(* IEC 61131-3 sources: plc-home-automation/home_automation/lighting_heating_updated/src/alarm, 4 files *)

(* ---- AlarmGlobals.st ---- *)
VAR_GLOBAL CONSTANT

   C_FRONT_DOOR_OPENING : INT     := 1;
   C_GARAGE_DOOR_OPENING : UINT   := 2;
   C_HALL_ZONE : UINT             := 4;
   C_GARAGE_ZONE : UINT           := 5;
   C_KITCHEN_ZONE : UINT          := 6;
   C_LIVING_ROOM_ZONE : UINT      := 7;
   C_BEDROOM_ZONE : UINT          := 8;
   C_DOWNSTAIRS_BATH_ZONE : UINT  := 9;
   C_HALLWAY_ZONE : UINT          := 10;
   C_CHILDRENS_ROOM_3_ZONE : UINT := 11;
   C_CHILDRENS_ROOM_1_ZONE : UINT := 12;
   C_CHILDRENS_ROOM_2_ZONE : UINT := 13;
   C_UPSTAIRS_BATH_ZONE : UINT    := 14;
   C_WC_ZONE : UINT               := 15;
   C_BOILER_ZONE : UINT           := 16;

   C_UNCONNECTED_NO_OP : UINT     := 3;

   C_ALARM_ZONES : UINT           := 16;
END_VAR

VAR_GLOBAL
    PARADOX_COM : fbPAR_DIG_EVOsystem;
    PARADOX_DATA : T_PAR_DIG_EVO_SYSTEM_DATA;
    ALARM_ZONES_INACTIVITY : ARRAY [1 .. C_ALARM_ZONES] OF BOOL;
    ALARM_ZONES_SABOTAGE : ARRAY [1 .. C_ALARM_ZONES] OF BOOL;
    ALARM_ZONES_ERROR : ARRAY [1 .. C_ALARM_ZONES] OF BOOL;
    ALARM_ACTIVE : BOOL;

    PRESENCE_BASED_HEATING_CONTROL : BOOL   := true;
    PRESENCE_BASED_HOT_WATER_CONTROL : BOOL := true;
    PRESENCE_BASED_HEATING_ENABLE : BOOL    := false;
    PRESENCE_BASED_HOT_WATER_ENABLE : BOOL  := false;

    AWAY_TIMER: TON;

    TIME_AWAY_SHORT : TIME     := T#20m;
    TIME_AWAY_LONG : TIME      := T#60m;
    GONE_FOR_5_SECONDS : BOOL  := FALSE; // for debugging purposes
    GONE_FOR_5_MINUTES : BOOL  := FALSE;
    GONE_FOR_5_HOURS : BOOL    := FALSE;
    GONE_FOR_SHORT_TIME : BOOL := FALSE;
    GONE_FOR_LONG_TIME : BOOL  := FALSE;
END_VAR

FUNCTION awayFromHomeFor : bool
  VAR_INPUT
    awayFor : TIME;  (*Tell me if motion sensors are inactive for that time. Max is 20 days.*)
  END_VAR

  IF(AWAY_TIMER.ET < awayFor) THEN
    awayFromHomeFor := false;
  ELSE
    awayFromHomeFor := true;
  END_IF;

END_FUNCTION

(* ---- AlarmRead.st ---- *)
FUNCTION alarmRead : BOOL

VAR_INPUT
END_VAR

VAR
  inactive_no_operation : BOOL := TRUE;
END_VAR

  PARADOX_COM(chan_code := CH1_uni, max_zone_count := C_ALARM_ZONES, par_system_data := PARADOX_DATA);
  alarmRead := PARADOX_COM.com_ok;

  ALARM_ZONES_INACTIVITY[C_FRONT_DOOR_OPENING] := PARADOX_DATA.zone[C_FRONT_DOOR_OPENING].state;
  ALARM_ZONES_INACTIVITY[C_GARAGE_DOOR_OPENING] := PARADOX_DATA.zone[C_GARAGE_DOOR_OPENING].state;
  ALARM_ZONES_INACTIVITY[C_HALL_ZONE] := PARADOX_DATA.zone[C_HALL_ZONE].state;
  ALARM_ZONES_INACTIVITY[C_GARAGE_ZONE] := PARADOX_DATA.zone[C_GARAGE_ZONE].state;
  ALARM_ZONES_INACTIVITY[C_KITCHEN_ZONE] := PARADOX_DATA.zone[C_KITCHEN_ZONE].state;
  ALARM_ZONES_INACTIVITY[C_LIVING_ROOM_ZONE] := PARADOX_DATA.zone[C_LIVING_ROOM_ZONE].state;
  ALARM_ZONES_INACTIVITY[C_BEDROOM_ZONE] := PARADOX_DATA.zone[C_BEDROOM_ZONE].state;
  ALARM_ZONES_INACTIVITY[C_DOWNSTAIRS_BATH_ZONE] := PARADOX_DATA.zone[C_DOWNSTAIRS_BATH_ZONE].state;
  ALARM_ZONES_INACTIVITY[C_HALLWAY_ZONE] := PARADOX_DATA.zone[C_HALLWAY_ZONE].state;
  ALARM_ZONES_INACTIVITY[C_CHILDRENS_ROOM_3_ZONE] := PARADOX_DATA.zone[C_CHILDRENS_ROOM_3_ZONE].state;
  ALARM_ZONES_INACTIVITY[C_CHILDRENS_ROOM_1_ZONE] := PARADOX_DATA.zone[C_CHILDRENS_ROOM_1_ZONE].state;
  ALARM_ZONES_INACTIVITY[C_CHILDRENS_ROOM_2_ZONE] := PARADOX_DATA.zone[C_CHILDRENS_ROOM_2_ZONE].state;
  ALARM_ZONES_INACTIVITY[C_UPSTAIRS_BATH_ZONE] := PARADOX_DATA.zone[C_UPSTAIRS_BATH_ZONE].state;
  ALARM_ZONES_INACTIVITY[C_WC_ZONE] := PARADOX_DATA.zone[C_WC_ZONE].state;
  ALARM_ZONES_INACTIVITY[C_BOILER_ZONE] := PARADOX_DATA.zone[C_BOILER_ZONE].state;

  ALARM_ZONES_SABOTAGE[C_FRONT_DOOR_OPENING] := PARADOX_DATA.zone[C_FRONT_DOOR_OPENING].tamper;
  ALARM_ZONES_SABOTAGE[C_GARAGE_DOOR_OPENING] := PARADOX_DATA.zone[C_GARAGE_DOOR_OPENING].tamper;
  ALARM_ZONES_SABOTAGE[C_HALL_ZONE] := PARADOX_DATA.zone[C_HALL_ZONE].tamper;
  ALARM_ZONES_SABOTAGE[C_GARAGE_ZONE] := PARADOX_DATA.zone[C_GARAGE_ZONE].tamper;
  ALARM_ZONES_SABOTAGE[C_KITCHEN_ZONE] := PARADOX_DATA.zone[C_KITCHEN_ZONE].tamper;
  ALARM_ZONES_SABOTAGE[C_LIVING_ROOM_ZONE] := PARADOX_DATA.zone[C_LIVING_ROOM_ZONE].tamper;
  ALARM_ZONES_SABOTAGE[C_BEDROOM_ZONE] := PARADOX_DATA.zone[C_BEDROOM_ZONE].tamper;
  ALARM_ZONES_SABOTAGE[C_DOWNSTAIRS_BATH_ZONE] := PARADOX_DATA.zone[C_DOWNSTAIRS_BATH_ZONE].tamper;
  ALARM_ZONES_SABOTAGE[C_HALLWAY_ZONE] := PARADOX_DATA.zone[C_HALLWAY_ZONE].tamper;
  ALARM_ZONES_SABOTAGE[C_CHILDRENS_ROOM_3_ZONE] := PARADOX_DATA.zone[C_CHILDRENS_ROOM_3_ZONE].tamper;
  ALARM_ZONES_SABOTAGE[C_CHILDRENS_ROOM_1_ZONE] := PARADOX_DATA.zone[C_CHILDRENS_ROOM_1_ZONE].tamper;
  ALARM_ZONES_SABOTAGE[C_CHILDRENS_ROOM_2_ZONE] := PARADOX_DATA.zone[C_CHILDRENS_ROOM_2_ZONE].tamper;
  ALARM_ZONES_SABOTAGE[C_UPSTAIRS_BATH_ZONE] := PARADOX_DATA.zone[C_UPSTAIRS_BATH_ZONE].tamper;
  ALARM_ZONES_SABOTAGE[C_WC_ZONE] := PARADOX_DATA.zone[C_WC_ZONE].tamper;
  ALARM_ZONES_SABOTAGE[C_BOILER_ZONE] := PARADOX_DATA.zone[C_BOILER_ZONE].tamper;

  ALARM_ZONES_ERROR[C_FRONT_DOOR_OPENING] := PARADOX_DATA.zone[C_FRONT_DOOR_OPENING].fault;
  ALARM_ZONES_ERROR[C_GARAGE_DOOR_OPENING] := PARADOX_DATA.zone[C_GARAGE_DOOR_OPENING].fault;
  ALARM_ZONES_ERROR[C_HALL_ZONE] := PARADOX_DATA.zone[C_HALL_ZONE].fault;
  ALARM_ZONES_ERROR[C_GARAGE_ZONE] := PARADOX_DATA.zone[C_GARAGE_ZONE].fault;
  ALARM_ZONES_ERROR[C_KITCHEN_ZONE] := PARADOX_DATA.zone[C_KITCHEN_ZONE].fault;
  ALARM_ZONES_ERROR[C_LIVING_ROOM_ZONE] := PARADOX_DATA.zone[C_LIVING_ROOM_ZONE].fault;
  ALARM_ZONES_ERROR[C_BEDROOM_ZONE] := PARADOX_DATA.zone[C_BEDROOM_ZONE].fault;
  ALARM_ZONES_ERROR[C_DOWNSTAIRS_BATH_ZONE] := PARADOX_DATA.zone[C_DOWNSTAIRS_BATH_ZONE].fault;
  ALARM_ZONES_ERROR[C_HALLWAY_ZONE] := PARADOX_DATA.zone[C_HALLWAY_ZONE].fault;
  ALARM_ZONES_ERROR[C_CHILDRENS_ROOM_3_ZONE] := PARADOX_DATA.zone[C_CHILDRENS_ROOM_3_ZONE].fault;
  ALARM_ZONES_ERROR[C_CHILDRENS_ROOM_1_ZONE] := PARADOX_DATA.zone[C_CHILDRENS_ROOM_1_ZONE].fault;
  ALARM_ZONES_ERROR[C_CHILDRENS_ROOM_2_ZONE] := PARADOX_DATA.zone[C_CHILDRENS_ROOM_2_ZONE].fault;
  ALARM_ZONES_ERROR[C_UPSTAIRS_BATH_ZONE] := PARADOX_DATA.zone[C_UPSTAIRS_BATH_ZONE].fault;
  ALARM_ZONES_ERROR[C_WC_ZONE] := PARADOX_DATA.zone[C_WC_ZONE].fault;
  ALARM_ZONES_ERROR[C_BOILER_ZONE] := PARADOX_DATA.zone[C_BOILER_ZONE].fault;

  ALARM_ZONES_INACTIVITY[C_UNCONNECTED_NO_OP] := inactive_no_operation;
  ALARM_ZONES_SABOTAGE[C_UNCONNECTED_NO_OP] := inactive_no_operation;
  ALARM_ZONES_ERROR[C_UNCONNECTED_NO_OP] := inactive_no_operation;

  ALARM_ACTIVE := PARADOX_DATA.part[1].state.armed;

  return;

END_FUNCTION

(* ---- Alarm.st ---- *)
PROGRAM AlarmControl
  VAR_INPUT
  END_VAR
  VAR_OUTPUT
  END_VAR
  VAR
     i: UINT;
     sumActivity : BOOL := FALSE;

     requestOffHeating : BOOL;
     requestOffHotWater : BOOL;

     heatingControl : ChangeOnOff;
     hotWaterControl : ChangeOnOff;

     heatingControllerName : STRING := 'Alarm heating control';
     hotWaterControllerName : STRING := 'Alarm hot water control';
  END_VAR

  alarmRead();

  // Turn on warm water circulation when someone enters through the entrance doors after the alarm cooldown time.
  VIRTUAL_CIRCULATION_SWITCH_IN := GONE_FOR_SHORT_TIME AND
      (NOT ALARM_ZONES_INACTIVITY[C_GARAGE_DOOR_OPENING] OR NOT ALARM_ZONES_INACTIVITY[C_FRONT_DOOR_OPENING]);

  // Detecting if house is no longer occupied or everyone is sleeping
  sumActivity := FALSE;
  FOR i := 1 TO C_ALARM_ZONES DO
     sumActivity := sumActivity OR (NOT ALARM_ZONES_INACTIVITY[i]);
  END_FOR;
  AWAY_TIMER(IN := NOT sumActivity, PT := T#20d);
  GONE_FOR_5_SECONDS  := awayFromHomeFor(awayFor := T#5s);
  GONE_FOR_5_MINUTES  := awayFromHomeFor(awayFor := T#5m);
  GONE_FOR_5_HOURS    := awayFromHomeFor(awayFor := T#5h);
  GONE_FOR_SHORT_TIME := awayFromHomeFor(TIME_AWAY_SHORT);
  GONE_FOR_LONG_TIME  := awayFromHomeFor(TIME_AWAY_LONG);

  requestOffHeating := ((ALARM_ACTIVE AND GONE_FOR_5_MINUTES) OR GONE_FOR_5_HOURS);
  requestOffHotWater:= ((ALARM_ACTIVE AND GONE_FOR_5_MINUTES) OR GONE_FOR_SHORT_TIME);

  IF PRESENCE_BASED_HEATING_CONTROL THEN
     heatingControl(requestOn := NOT requestOffHeating,
         requestOff := requestOffHeating,
         name := heatingControllerName);
     PRESENCE_BASED_HEATING_ENABLE := heatingControl.output;
  END_IF;

  IF PRESENCE_BASED_HOT_WATER_CONTROL THEN
     hotWaterControl(requestOn := NOT requestOffHotWater,
         requestOff := requestOffHotWater,
         name := hotWaterControllerName);
     PRESENCE_BASED_HOT_WATER_ENABLE := hotWaterControl.output;
  END_IF;

END_PROGRAM

(* ---- AlarmInit.st ---- *)
PROGRAM AlarmInit
  VAR_INPUT
  END_VAR
  VAR_OUTPUT
  END_VAR
  VAR
  END_VAR
  VAR_TEMP
  END_VAR

VAR
  initialised : BOOL := FALSE;
END_VAR;

    IF initialised = FALSE THEN
        initialised := TRUE;
    ELSE
        // No opeartion
    END_IF;

END_PROGRAM
